// TIA Portal V16 export
// export: Created 2022-11-17T15:49:36.15724Z, ExportSetting WithDefaults, DisplayName Totally Integrated Automation Portal, DisplayVersion V16 Update 6, DisplayName TIA Portal Version Control Interface, DisplayVersion V16 Update 2, DisplayName TIA Portal Openness, DisplayVersion V16 Update 6, DisplayName SINAMICS Startdrive Advanced, DisplayVersion V16 Update 5, DisplayName SINAMICS Startdrive G130, G150, S120, S150, SINAMICS MV, S210, DisplayVersion V16 Update 5, DisplayName SINAMICS Startdrive G110M, G120, G120C, G120D, G120P, G115D, DisplayVersion V16 Update 5, DisplayName STEP 7 Professional, DisplayVersion V16 Update 6, DisplayName STEP 7 Safety, DisplayVersion V16, DisplayName WinCC Advanced, DisplayVersion V16 Update 6
DATA_BLOCK "DB03_Machine"   // DB3
{ S7_Optimized_Access := 'FALSE' }
AUTHOR : Robopac
VERSION : 0.0
// stored: AutoNumber false, IsOnlyStoredInLoadMemory false, IsWriteProtectedInAS false
   VAR RETAIN
      dbx0_0 : Bool := FALSE;   // Enable the arm rotation revolution counter
      dbx0_1 : Bool := FALSE;   // High pressure on prestretch roller dancer
      dbx0_2 : Bool := FALSE;   // One arm revolution done support memory
      dbx0_3 : Bool := FALSE;   // One arm revolution done
      dbx0_4 : Bool := FALSE;   // Support memory for revolution counter
      dbx0_5 : Bool := FALSE;   // Support memory for 10% prestretch carriage
      dbx0_6 : Bool := FALSE;
      dbx0_7 : Bool := FALSE;   // Support memory for arm rotation speed recorded
      dbb1 : Byte := 16#00;
      MachineExc : Bool := FALSE;   // Wrapping excluded
      MachineInc : Bool := FALSE;   // Wrapping included
      dbb3 : Byte := 16#00;
      dbx4_0 : Bool := FALSE;   // Memory to silent acoustic signal on alarm
      dbx4_1 : Bool := FALSE;
      dbx4_2 : Bool := FALSE;   // Condition to check all out of positon alarm
      dbx4_3 : Bool := FALSE;   // Condition for manual operation
      dbx4_4 : Bool := FALSE;   // All units are ready for automatic cycle
      dbx4_5 : Bool := FALSE;
      dbx4_6 : Bool := FALSE;   // Data for next ring height loaded
      dbx4_7 : Bool := FALSE;   // Data for next ring height loaded
      dbx5_0 : Bool := FALSE;   // Wrapping cycle: Next step is cut and pallet unload
      dbx5_1 : Bool := FALSE;   // Wrapping cycle: Next step is cut and new spool carriage height
      dbx5_2 : Bool := FALSE;   // Wrapping cycle: Next step is new spool carriage height
      dbx5_3 : Bool := FALSE;   // Wrapping cycle: After this step top waterproof
      dbx5_4 : Bool := FALSE;   // Wrong data program for the pallet on the machine
      dbx5_5 : Bool := FALSE;   // Closing upper(double) rope unit
      dbx5_6 : Bool := FALSE;   // Closing single or lower(double) rope unit
      dbx5_7 : Bool := FALSE;   // Memory for timeout enable
      dbx6_0 : Bool := FALSE;   // Memory to exclude infeed safety barrier
      dbx6_1 : Bool := FALSE;   // Memory to exclude outfeed safety barrier
      dbx6_2 : Bool := FALSE;   // Memory to exclude infeed safety barrier
      dbx6_3 : Bool := FALSE;   // Memory to exclude infeed safety barrier
      dbx6_4 : Bool := FALSE;   // Memory to exclude outfeed safety barrier
      dbx6_5 : Bool := FALSE;   // Memory to exclude outfeed safety barrier
      dbx6_6 : Bool := FALSE;
      dbx6_7 : Bool := FALSE;
      dbx7_0 : Bool := FALSE;   // Pressure plate excluded for low pallet
      dbx7_1 : Bool := FALSE;
      dbx7_2 : Bool := FALSE;   // Support memory to check rotation speed
      dbx7_3 : Bool := FALSE;   // Support memory to check spool carriage speed
      dbx7_4 : Bool := FALSE;   // Used by S7-200
      dbx7_5 : Bool := FALSE;   // Machine in wrapping cycle
      dbx7_6 : Bool := FALSE;   // Support memory to refresh pallet per hour value
      dbx7_7 : Bool := FALSE;
      dbb8 : Byte := 16#00;
      TopExc : Bool := FALSE;   // Top excluded
      TopBefore : Bool := FALSE;   // Top included before wrapping beginning
      TopWaterP : Bool := FALSE;   // Top included waterproof
      dbw10 : Int := 0;
      dbw12 : Int := 0;   // Counter for revolution on running spool carriage height
      dbw14 : Int := 0;   // Counter for revolution on welder contrast
      dbw16 : Int := 0;   // Counter for revolution of deceleration
      dbw18 : Int := 0;
      dbw20 : Int := 0;   // Active program for multiprogram (Display)
      dbw22 : Int := 0;   // Selected program for multiprogram (Display)
      dbw24 : Int := 0;   // Program to be shown on data program page (Display)
      dbw26 : Int := 0;   // Program selection by external signal
      dbw28 : Int := 0;   // Program selection by external signal
      dbw30 : Int := 0;   // Support memory for data transfer
      dbw32 : Int := 0;   // Arm rotation speed recorded (rpm*10)
      dbw34 : Int := 0;   // Required arm rotation speed recorded (%*10)
      dbw36 : Int := 0;
      dbw38 : Int := 0;   // Support memory to evaluate carriage movement speed
      dbw40 : Int := 0;   // Support memory to evaluate carriage movement speed
      dbw42 : Int := 0;   // Spool carriage movement speed mm/sec
      dbw44 : Int := 0;   // table rotation movement speed mm/sec
      dbw46 : Int := 0;   // Arm rotation speed (rpm*10) related to actual required speed
      dbw48 : Int := 0;   // Spool carriage movement speed mm/sec recorded
      dbw50 : Int := 0;
      dbw52 : Int := 0;   // High speed for spool carriage movement (%) recorded from display
      dbw54 : Int := 0;   // upport memory for spool carriage high speed
      dbw56 : Int := 0;   // Spool carriage movement speed used on cycle (mm/sec)
      dbb58 : Byte := 16#00;   // Counter for DAC M20 converter
      dbx59_0 : Bool := FALSE;   // Arm rotation and top carriage speed change for DAC M20
      dbx59_1 : Bool := FALSE;   // Spool carriage speed change for DAC M20
      dbx59_2 : Bool := FALSE;   // Counter for DAC M20 is odd
      dbx59_3 : Bool := FALSE;
      dbx59_4 : Bool := FALSE;
      dbx59_5 : Bool := FALSE;
      dbx59_6 : Bool := FALSE;
      dbx59_7 : Bool := FALSE;
      dbw60 : Int := 0;   // Value for DAC analog output
      dbw62 : Int := 0;
      dbw64 : Int := 0;
      dbw66 : Int := 0;   // Support for running height data transfer
      dbw68 : Int := 0;   // Number of the running spool carriage height
      dbw70 : Int := 0;   // Film overlap for running spool carriage height
      dbw72 : Int := 0;   // Carriage height (mm) for running spool carriage height
      dbx74_0 : Bool := FALSE;   // Landmark (0=Bottom 1=Top) for running spool carriage height
      dbx74_1 : Bool := FALSE;   // Pallet lifter for running spool carriage height (0=Excluded 1=Included)
      dbx74_2 : Bool := FALSE;   // Spare
      dbx74_3 : Bool := FALSE;   // Airblower on film tail for running spool carriage height (0=Exc 1=Inc)
      dbx74_4 : Bool := FALSE;   // Next step for running spool carriage height (0=End 1=Next)
      dbx74_5 : Bool := FALSE;   // Pressure plate for running spool carriage height (0=Excluded 1=Included)
      dbx74_6 : Bool := FALSE;   // Spare
      dbx74_7 : Bool := FALSE;   // Spare
      dbb75 : Byte := 16#00;   // Spare
      dbw76 : Int := 0;   // Revolutions for running spool carriage height
      dbb78 : Byte := 16#00;   // Rope unit for running spool carriage height (1=Excluded 2=Inc 3=Inc during)
      dbb79 : Byte := 16#00;   // Rope unit for running spool carriage height (1=Excluded 2=Inc 3=Inc during)
      dbw80 : Int := 0;   // Film force for running spool carriage height
      dbw82 : Int := 0;   // Film prestretch for running spool carriage height
      dbw84 : Int := 0;   // Delay to open or close upper rope unit for runninh spool carriage height
      dbw86 : Int := 0;   // Delay to open or close lower rope unit for runninh spool carriage height
      dbw88 : Int := 0;   // Spare for running spool carriage height
      dbw90 : Int := 0;   // Spare for running spool carriage height
      dbw92 : Int := 0;   // Spare for running spool carriage height
      dbw94 : Int := 0;   // Spare for running spool carriage height
      dbw96 : Int := 0;
      dbw98 : Int := 0;
   END_VAR
BEGIN
END_DATA_BLOCK
